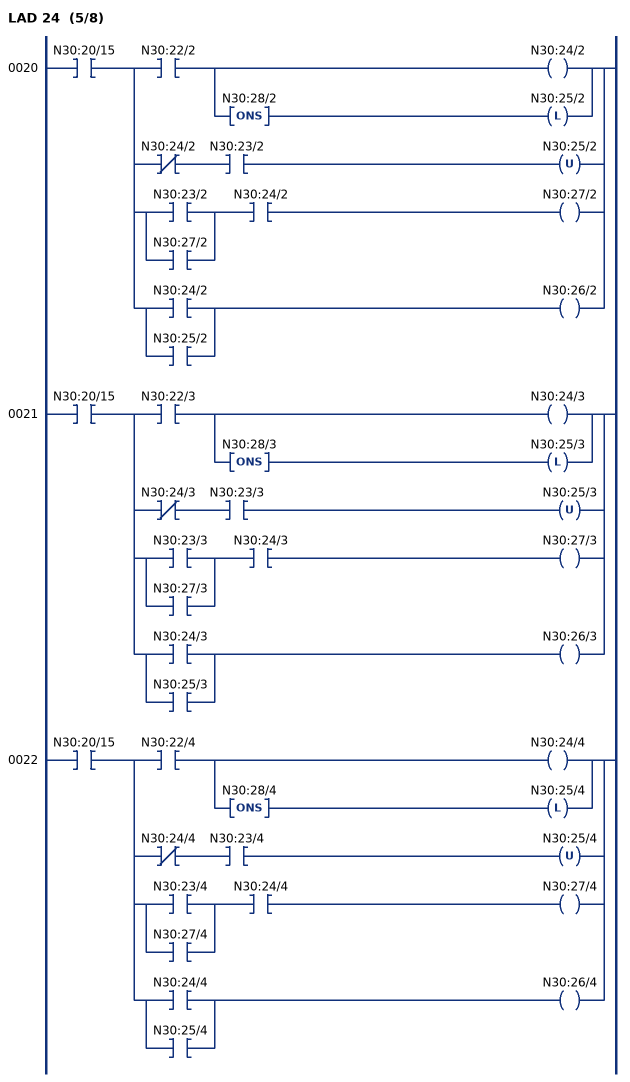
% Rung: 20 %
SOR XIC N30:20/15 BST XIC N30:22/2 BST OTE N30:24/2 NXB OSR N30:28/2 OTL N30:25/2 BND NXB XIO N30:24/2 XIC N30:23/2 OTU N30:25/2 NXB BST XIC N30:23/2 NXB XIC N30:27/2 BND XIC N30:24/2 OTE N30:27/2 NXB BST XIC N30:24/2 NXB XIC N30:25/2 BND OTE N30:26/2 BND EOR
% Rung: 21 %
SOR XIC N30:20/15 BST XIC N30:22/3 BST OTE N30:24/3 NXB OSR N30:28/3 OTL N30:25/3 BND NXB XIO N30:24/3 XIC N30:23/3 OTU N30:25/3 NXB BST XIC N30:23/3 NXB XIC N30:27/3 BND XIC N30:24/3 OTE N30:27/3 NXB BST XIC N30:24/3 NXB XIC N30:25/3 BND OTE N30:26/3 BND EOR
% Rung: 22 %
SOR XIC N30:20/15 BST XIC N30:22/4 BST OTE N30:24/4 NXB OSR N30:28/4 OTL N30:25/4 BND NXB XIO N30:24/4 XIC N30:23/4 OTU N30:25/4 NXB BST XIC N30:23/4 NXB XIC N30:27/4 BND XIC N30:24/4 OTE N30:27/4 NXB BST XIC N30:24/4 NXB XIC N30:25/4 BND OTE N30:26/4 BND EOR

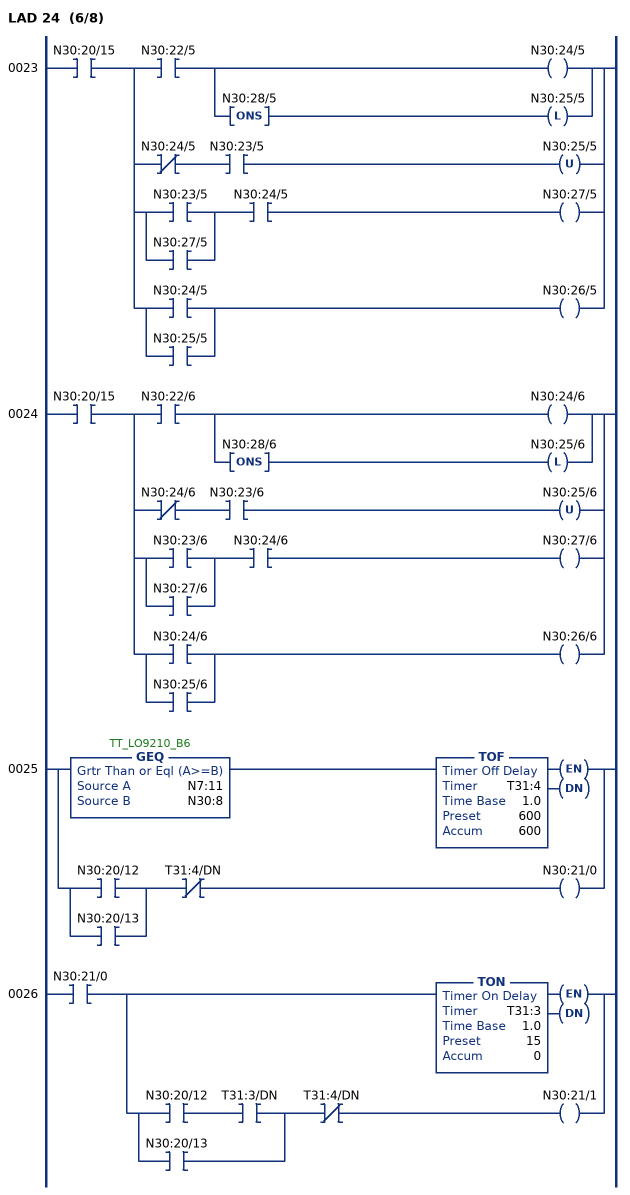
% Rung: 23 %
SOR XIC N30:20/15 BST XIC N30:22/5 BST OTE N30:24/5 NXB OSR N30:28/5 OTL N30:25/5 BND NXB XIO N30:24/5 XIC N30:23/5 OTU N30:25/5 NXB BST XIC N30:23/5 NXB XIC N30:27/5 BND XIC N30:24/5 OTE N30:27/5 NXB BST XIC N30:24/5 NXB XIC N30:25/5 BND OTE N30:26/5 BND EOR
% Rung: 24 %
SOR XIC N30:20/15 BST XIC N30:22/6 BST OTE N30:24/6 NXB OSR N30:28/6 OTL N30:25/6 BND NXB XIO N30:24/6 XIC N30:23/6 OTU N30:25/6 NXB BST XIC N30:23/6 NXB XIC N30:27/6 BND XIC N30:24/6 OTE N30:27/6 NXB BST XIC N30:24/6 NXB XIC N30:25/6 BND OTE N30:26/6 BND EOR
% Rung: 25 %
SOR BST GEQ N7:11 N30:8 TOF T31:4 1.0 600 600 NXB BST XIC N30:20/12 NXB XIC N30:20/13 BND XIO T31:4/DN OTE N30:21/0 BND EOR
%   N7:11  TT_LO9210_B6 %
% Rung: 26 %
SOR XIC N30:21/0 BST TON T31:3 1.0 15 0 NXB BST XIC N30:20/12 XIC T31:3/DN NXB XIC N30:20/13 BND XIO T31:4/DN OTE N30:21/1 BND EOR

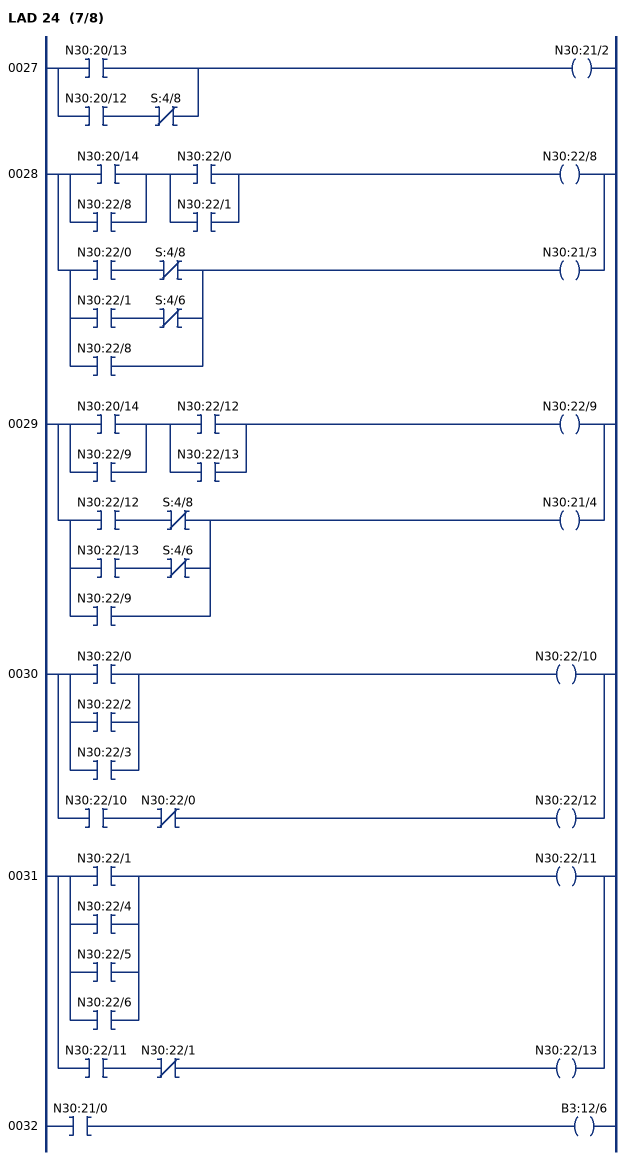
% Rung: 27 %
SOR BST XIC N30:20/13 NXB XIC N30:20/12 XIO S:4/8 BND OTE N30:21/2 EOR
% Rung: 28 %
SOR BST BST XIC N30:20/14 NXB XIC N30:22/8 BND BST XIC N30:22/0 NXB XIC N30:22/1 BND OTE N30:22/8 NXB BST XIC N30:22/0 XIO S:4/8 NXB XIC N30:22/1 XIO S:4/6 NXB XIC N30:22/8 BND OTE N30:21/3 BND EOR
% Rung: 29 %
SOR BST BST XIC N30:20/14 NXB XIC N30:22/9 BND BST XIC N30:22/12 NXB XIC N30:22/13 BND OTE N30:22/9 NXB BST XIC N30:22/12 XIO S:4/8 NXB XIC N30:22/13 XIO S:4/6 NXB XIC N30:22/9 BND OTE N30:21/4 BND EOR
% Rung: 30 %
SOR BST BST XIC N30:22/0 NXB XIC N30:22/2 NXB XIC N30:22/3 BND OTE N30:22/10 NXB XIC N30:22/10 XIO N30:22/0 OTE N30:22/12 BND EOR
% Rung: 31 %
SOR BST BST XIC N30:22/1 NXB XIC N30:22/4 NXB XIC N30:22/5 NXB XIC N30:22/6 BND OTE N30:22/11 NXB XIC N30:22/11 XIO N30:22/1 OTE N30:22/13 BND EOR
% Rung: 32 %
SOR XIC N30:21/0 OTE B3:12/6 EOR

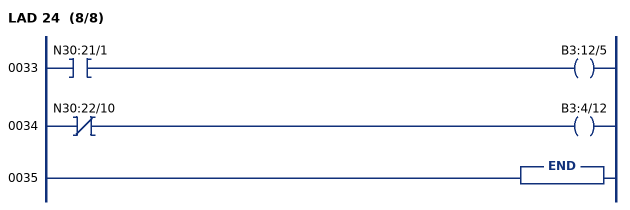
% Rung: 33 %
SOR XIC N30:21/1 OTE B3:12/5 EOR
% Rung: 34 %
SOR XIO N30:22/10 OTE B3:4/12 EOR
% Rung: 35 %
SOR END EOR

OTHER DOCUMENTED ADDRESSES
  11QM1  "Thermique moteur"
  B3:2/3  P9211_A_TOURNER
  B3:2/4  P9212_A_TOURNER
  B3:3/0  SET_RESET_REMPLISSAG  "SET ET RESET LE REMPLISSAGE CUVE EDI"
  B3:3/9  XV_LO9230A6  "Vanne retour boucle"
  B3:4/4  AU_ENCLENCHER
  B3:4/5  RESET_AU
  B3:4/15  STRESS
  B13:4/0  OSR_START_SANIT
  DFILE:0  "OUTPUT"
  DFILE:1  "INPUT"
  DFILE:2  "STATUS"
  DFILE:3  "BINARY"
  DFILE:4  "TIMER"
  DFILE:5  "COUNTER"
  DFILE:6  "CONTROL"
  DFILE:7  "INTEGER"
  DFILE:8  "FLOAT"
  DFILE:9  "PID REFROI"
  DFILE:10  "PARA"
  DFILE:13  "BIN SANIT"
  DFILE:14  "TIMER SANI"
  DFILE:17  "INT SANIT"
  DFILE:19  "PID CHAUFF"
  DFILE:20  "PARA SANIT"
  N7:7  AI1_RESERVE
  N7:27  PASSWORD
  N7:28  PAGE
  N7:68/0  AL1_P9211  "Pompe P9211 en défaut (masqué)"
  N7:68/1  AL1_P9212  "Pompe P9212 en défaut (masqué)"
  N7:68/2  AL1_ZERO_SELECT  "Pas de sélection Sanitisation / production (masqué)"
  N9:3  TC_LO9200A8_KP  "Gain de la régulation de température"
  N9:4  TC_LO9200A8_TI  "intégrale"
  N9:5  TC_LO9200A8_TD  "Dérivée"
  N9:6  BIAS_FROID
  N9:8  SETPOINT_MINI_FROID
  N9:11  OUT_MAX_FROID
  N9:12  OUT_MIN_FROID
  N19:3  TC_LO9200B8_KP  "Gain de la régulation de température"
  N19:4  TC_LO9200B8_TI  "intégrale"
  N19:5  TC_LO9200B8_TD  "Dérivée"
  N19:6  BIAS_CHAUFF
  N19:8  SETPOINT_MINI_CHAUFF
  N19:11  OUT_MAX_CHAUFF
  N19:12  OUT_MIN_CHAUFF
  PFILE:3  "Table d'entrée"
  PFILE:6  "PRODUCTION EDI"
  PFILE:7  "SANITISATION"
  PFILE:8  "GESTION DES AFFICHAG E"
  PFILE:10  "REMPLISSAGE DE LA CU VE"
  PFILE:11  "GESTION DES UNITEE U V"
  PFILE:12  "REGULATION DE REFROI DIR"
  PFILE:13  "GESTION DE LA CONDUC TIVITE"
  PFILE:14  "INTEDICTION DE SORTI E DE L EDI"
  PFILE:15  "GESTION DES POMPES"
  PFILE:22  "REGULATION DE CHAUFF ER"
  Q21:0  ETAP0
  Q21:1  ETAP1
  Q21:2  ETAP2
  Q21:3  ETAP3
  Q21:4  ETAP4
  Q21:5  ETAP5
  Q21:6  ETAP6
  Q21:7  ETAP7
  Q21:8  ETAP8
  Q21:9  ETAP9
  Q21:10  ETAP10
  Q21:11  ETAP11
  Q21:12  ETAP12
  Q21:13  ETAP13
  T4:0/DN  "Tempo d'autorisation washer"

COMMENTS NOT ATTACHED TO A CURRENT RUNG
  T4:9: OUT OF RANGEMESURE DE TEMPERATURE
  N7:64/0: Alarme de niveau 3
  T4:1: Alarme de niveau 2
  O:6.0/0: Carte de sortie digitale N°6
  N7:0: AIT LO9230 A2 ( Conductivité EDI Boucle)
  N7:12: LT VS9210A3 Niveau de la cuve
  N7:8: TIT LO9230A3 TEMPERATURE DE BOUCLE
  N7:4: RESERVE
  T4:6: Out of range mesure de niveau
    Alarme N°
  T4:8: OUT OF RANGE MESURE DE CONDUCTIVITE
  N7:67: Etablissement des masques pour les alarmes toujours active
  U:5: Alarmes
  T4:18: Alarme N°1
  T4:21: Alarme de niveau 3
  N7:64/1: Alarme N°10
  N7:62/6: Alarme N°10

REVISION NOTES
  1: Correction blocage du niveau à zéro (demande de P. Vandersand (BV2)

DATA TABLE (non-zero values as saved)
DATA B3
% B3:0 % 0X7029 0X0889 0X0110 0X0004 0X1000 0X0080 0X0000 0X0001 0X0110 0X016F
% B3:10 % 0X0000 0X0006 0X0000 0X0000 0X0000 0X0000 0X0000 0X0000 0X0000 0X0000
DATA T4
% .PRE .ACC %
% T4:0 % 32766 0
% T4:1 % 5 5
% T4:2 % 5 5
% T4:3 % 5 0
% T4:4 % 30 0
% T4:5 % 120 120
% T4:6 % 5 0
% T4:7 % 5 0
% T4:8 % 5 0
% T4:9 % 5 0
% T4:10 % 5 0
% T4:11 % 5 5
% T4:12 % 5 0
% T4:13 % 5 5
% T4:14 % 5 0
% T4:15 % 5 0
% T4:16 % 5 0
% T4:17 % 5 0
% T4:18 % 5 0
% T4:19 % 5 0
% T4:23 % 60 0
% T4:24 % 60 0
% T4:25 % 2 0
% T4:26 % 10 0
% T4:27 % 1 0
% T4:28 % 5 0
% T4:29 % 5 0
% T4:30 % 32700 0
% T4:31 % 32767 0
% T4:32 % 5 0
% T4:33 % 5 0
DATA N7
% N7:0 % 0 0 400 44 0 0 1000 -242 1 0
% N7:10 % 1500 294 1 0 28000 0 27000 25000 24000 9000
% N7:20 % 6000 5000 240 0 100 110 100 1 1 0
% N7:30 % 0 35 0 0 0 0 0 0 0 0
% N7:60 % 4 7 19 0 8 2 160 13 4 0
% N7:70 % 0 0 0 0 0 20 0 0 0 0
% N7:80 % 7634 0 0 0 0 0 0 0 0 0
DATA N9
% N9:0 % 12 0 150 250 2 4 0 16383 0 0
% N9:10 % 0 100 0 1 150 0 49 0 0 0
% N9:20 % 0 0 150 0
DATA N10
% N10:0 % 0 0 400 0 1500 0 28000 30 60 0
% N10:10 % 100 250 100 250 0 900 750 900 150
DATA B13
% B13:0 % 0X0D00 0X0000 0X0000 0X0000 0XC000 0X0000 0X0000 0X0000 0X0000 0X007F
DATA T14
% .PRE .ACC %
% T14:0 % 5 0
% T14:1 % 5 0
% T14:2 % 5 0
% T14:3 % 240 0
% T14:4 % 5 0
% T14:5 % 7200 0
% T14:6 % 60 0
% T14:7 % 5 0
% T14:8 % 5 0
% T14:9 % 5 0
% T14:10 % 5 5
% T14:11 % 5 5
% T14:12 % 5 0
% T14:13 % 9000 0
% T14:14 % 3600 0
% T14:15 % 5 0
% T14:16 % 5 0
% T14:17 % 300 0
% T14:18 % 35 0
% T14:19 % 5 0
% T14:20 % 5 0
DATA N17
% N17:0 % 0 0 0 1500 246 -250 250 7 0 1000
% N17:10 % 220 150 560 750 900 850 0 0 0 0
% N17:30 % 0 150 0 0 0 0 0 0 0 0
% N17:40 % 781 0 0 0 0 0 0 0 0 0
DATA N19
% N19:0 % 8 0 810 200 2 6 0 16383 0 0
% N19:10 % 0 100 0 1 810 0 1 0 0 0
% N19:20 % 0 0 810 0
DATA N20
% N20:0 % 6500 0 1500 0 1000 -250 250 760 7200 -125
% N20:10 % 125
DATA N30
% N30:0 % 0 250 500 480 10 4 30 15 980 10
% N30:10 % 0 250 500 0 0 0 0 0 0 0
% N30:20 % 1031 0 0 0 0 0 0 0 0 0
DATA T31
% .PRE .ACC %
% T31:0 % 28800 0
% T31:1 % 10 10
% T31:2 % 1800 0
% T31:3 % 15 0
% T31:4 % 600 600
